DATA_BLOCK "DIH"
{ S7_Optimized_Access := 'FALSE' }
VERSION : 0.1
NON_RETAIN
   STRUCT
      HAD10_AA101_PWR : "DIVAR_HMI";   // Клапан неперевної продувки. (Контроль живлення) {CJF01}
      LAB10_AA001_PWR : "DIVAR_HMI";   // Регулятор рівня в барабані. (Контроль живлення) {CJF01}
      CJF01_SB001_ESTP : "DIVAR_HMI";   // СТОП Шафа SCPU {CJF01}
      CJF01_SB002_ESTP : "DIVAR_HMI";   // СТОП Шафа Пневмоострів {CJF01}
      REZDI_CJF01_MOD11_CH4 : "DIVAR_HMI";   // Резерв DI, рейка CJF01, модуль 11, канал 4 {CJF01}
      HCB10_AA601_SOPN : "DIVAR_HMI";   // Клапан Обдувного апарату №1 (Спрацювання) {CJF01}
      HCB20_AA601_SOPN : "DIVAR_HMI";   // Клапан Обдувного апарату №2 (Спрацювання) {CJF01}
      HCB30_AA601_SOPN : "DIVAR_HMI";   // Клапан Обдувного апарату №3 (Спрацювання) {CJF01}
      HCB40_AA601_SOPN : "DIVAR_HMI";   // Клапан Обдувного апарату №4 (Спрацювання) {CJF01}
      HCB50_AA601_SOPN : "DIVAR_HMI";   // Клапан Обдувного апарату №5 (Спрацювання) {CJF01}
      HCB60_AA601_SOPN : "DIVAR_HMI";   // Клапан Обдувного апарату №6 (Спрацювання) {CJF01}
      HCB70_AA601_SOPN : "DIVAR_HMI";   // Клапан Обдувного апарату №7 (Спрацювання) {CJF01}
      HCB80_AA601_SOPN : "DIVAR_HMI";   // Клапан Обдувного апарату №8 (Спрацювання) {CJF01}
      HCB90_AA601_SOPN : "DIVAR_HMI";   // Клапан Обдувного апарату №9 (Спрацювання) {CJF01}
      HCB100_AA601_SOPN : "DIVAR_HMI";   // Клапан Обдувного апарату №10 (Спрацювання) {CJF01}
      REZDI_CJF01_MOD11_CH15 : "DIVAR_HMI";   // Резерв DI, рейка CJF01, модуль 11, канал 15 {CJF01}
      HLA10_AA151_SOPN : "DIVAR_HMI";   // Шибер первинного повітря №1 (Відкритий) {CJF01}
      HLA10_AA151_SCLS : "DIVAR_HMI";   // Шибер первинного повітря №1 (Закритий) {CJF01}
      HLA10_AA152_SOPN : "DIVAR_HMI";   // Шибер первинного повітря №2 (Відкритий) {CJF01}
      HLA10_AA152_SCLS : "DIVAR_HMI";   // Шибер первинного повітря №2 (Закритий) {CJF01}
      HHB11_SOPN : "DIVAR_HMI";   // Колосники "Поле №1" (Відкритий) {CJF01}
      HHB11_SCLS : "DIVAR_HMI";   // Колосники "Поле №1" (Закритий) {CJF01}
      HHB12_SOPN : "DIVAR_HMI";   // Колосники "Поле №2" (Відкритий) {CJF01}
      HHB12_SCLS : "DIVAR_HMI";   // Колосники "Поле №2" (Закритий) {CJF01}
      HHB13_SOPN : "DIVAR_HMI";   // Колосники "Поле №3" (Відкритий) {CJF01}
      HHB13_SCLS : "DIVAR_HMI";   // Колосники "Поле №3" (Закритий) {CJF01}
      HHB14_SOPN : "DIVAR_HMI";   // Колосники "Поле №4" (Відкритий) {CJF01}
      HHB14_SCLS : "DIVAR_HMI";   // Колосники "Поле №4" (Закритий) {CJF01}
      REZDI_CJF01_MOD12_CH12 : "DIVAR_HMI";   // Резерв DI, рейка CJF01, модуль 12, канал 12 {CJF01}
      REZDI_CJF01_MOD12_CH13 : "DIVAR_HMI";   // Резерв DI, рейка CJF01, модуль 12, канал 13 {CJF01}
      REZDI_CJF01_MOD12_CH14 : "DIVAR_HMI";   // Резерв DI, рейка CJF01, модуль 12, канал 14 {CJF01}
      REZDI_CJF01_MOD12_CH15 : "DIVAR_HMI";   // Резерв DI, рейка CJF01, модуль 12, канал 15 {CJF01}
      HNC10_AF001_PWR : "DIVAR_HMI";   // Димосос ДН1 (Контроль живлення) {CJF06}
      HNC10_AF001_LSTP : "DIVAR_HMI";   // Димосос ДН1 (Кнопка стоп) {CJF06}
      HNC10_AF001_RUN : "DIVAR_HMI";   // Димосос ДН1 (Робота) {CJF06}
      HNC10_AF001_ALM : "DIVAR_HMI";   // Димосос ДН1 (Аварія ПЧ) {CJF06}
      HNC20_AF001_PWR : "DIVAR_HMI";   // Димосос ДН2 (Контроль живлення) {CJF06}
      HNC20_AF001_LSTP : "DIVAR_HMI";   // Димосос ДН2 (Кнопка стоп) {CJF06}
      HNC20_AF001_RUN : "DIVAR_HMI";   // Димосос ДН2 (Робота) {CJF06}
      HNC20_AF001_ALM : "DIVAR_HMI";   // Димосос ДН2 (Аварія ПЧ) {CJF06}
      HLA10_AF001_PWR : "DIVAR_HMI";   // Вентилятор первинного дуття ДВ1 (Контроль живлення) {CJF06}
      HLA10_AF001_LSTP : "DIVAR_HMI";   // Вентилятор первинного дуття ДВ1 (Кнопка стоп) {CJF06}
      HLA10_AF001_RUN : "DIVAR_HMI";   // Вентилятор первинного дуття ДВ1 (Робота) {CJF06}
      HLA10_AF001_ALM : "DIVAR_HMI";   // Вентилятор первинного дуття ДВ1 (Аварія ПЧ) {CJF06}
      HLA20_AF001_PWR : "DIVAR_HMI";   // Вентилятор вторинного дуття ДВ2 (Контроль живлення) {CJF06}
      HLA20_AF001_LSTP : "DIVAR_HMI";   // Вентилятор вторинного дуття ДВ2 (Кнопка стоп) {CJF06}
      HLA20_AF001_RUN : "DIVAR_HMI";   // Вентилятор вторинного дуття ДВ2 (Робота) {CJF06}
      HLA20_AF001_ALM : "DIVAR_HMI";   // Вентилятор вторинного дуття ДВ2 (Аварія ПЧ) {CJF06}
      LAB01_AP001_PWR : "DIVAR_HMI";   // Живильний насос №1 (Контроль живлення) {CJF06}
      LAB01_AP001_LSTP : "DIVAR_HMI";   // Живильний насос №1 (Кнопка стоп) {CJF06}
      LAB01_AP001_RUN : "DIVAR_HMI";   // Живильний насос №1 (Робота) {CJF06}
      LAB01_AP001_ALM : "DIVAR_HMI";   // Живильний насос №1 (Аварія ПЧ) {CJF06}
      LAB02_AP002_PWR : "DIVAR_HMI";   // Живильний насос №2 (Контроль живлення) {CJF06}
      LAB02_AP002_LSTP : "DIVAR_HMI";   // Живильний насос №2 (Кнопка стоп) {CJF06}
      LAB02_AP002_RUN : "DIVAR_HMI";   // Живильний насос №2 (Робота) {CJF06}
      LAB02_AP002_ALM : "DIVAR_HMI";   // Живильний насос №2 (Аварія ПЧ) {CJF06}
      HFB11_AF001_PWR : "DIVAR_HMI";   // Шнек подачі палива №1 (Контроль живлення) {CJF06}
      HFB11_AF001_LSTP : "DIVAR_HMI";   // Шнек подачі палива №1 (Кнопка стоп) {CJF06}
      HFB11_AF001_RUN : "DIVAR_HMI";   // Шнек подачі палива №1 (Робота) {CJF06}
      HFB11_AF001_ALM : "DIVAR_HMI";   // Шнек подачі палива №1 (Аварія ПЧ) {CJF06}
      HFB21_AF001_PWR : "DIVAR_HMI";   // Шнек подачі палива №2 (Контроль живлення) {CJF06}
      HFB21_AF001_LSTP : "DIVAR_HMI";   // Шнек подачі палива №2 (Кнопка стоп) {CJF06}
      HFB21_AF001_RUN : "DIVAR_HMI";   // Шнек подачі палива №2 (Робота) {CJF06}
      HFB21_AF001_ALM : "DIVAR_HMI";   // Шнек подачі палива №2 (Аварія ПЧ) {CJF06}
      HFB12_AF001_PWR : "DIVAR_HMI";   // Транспортер подачі палива №1 (Контроль живлення) {CJF06}
      HFB12_AF001_LSTP : "DIVAR_HMI";   // Транспортер подачі палива №1 (Кнопка стоп) {CJF06}
      HFB12_AF001_RUN : "DIVAR_HMI";   // Транспортер подачі палива №1 (Робота) {CJF06}
      HFB12_AF001_ALM : "DIVAR_HMI";   // Транспортер подачі палива №1 (Аварія ПЧ) {CJF06}
      HFB22_AF001_PWR : "DIVAR_HMI";   // Транспортер подачі палива №2 (Контроль живлення) {CJF06}
      HFB22_AF001_LSTP : "DIVAR_HMI";   // Транспортер подачі палива №2 (Кнопка стоп) {CJF06}
      HFB22_AF001_RUN : "DIVAR_HMI";   // Транспортер подачі палива №2 (Робота) {CJF06}
      HFB22_AF001_ALM : "DIVAR_HMI";   // Транспортер подачі палива №2 (Аварія ПЧ) {CJF06}
      EKG11_AF001_PWR : "DIVAR_HMI";   // Пульсатор (Контроль живлення) {CJF06}
      EKG11_AF001_LSTP : "DIVAR_HMI";   // Пульсатор (Кнопка стоп) {CJF06}
      EKG11_AF001_RUN : "DIVAR_HMI";   // Пульсатор (Робота) {CJF06}
      EKG11_AF001_ALM : "DIVAR_HMI";   // Пульсатор (Аварія ПЧ) {CJF06}
      Rez1_PWR : "DIVAR_HMI";   // Резервний привод ПЧ (Контроль живлення) {CJF06}
      Rez1_LSTP : "DIVAR_HMI";   // Резервний привод ПЧ (Кнопка стоп) {CJF06}
      Rez1_RUN : "DIVAR_HMI";   // Резервний привод ПЧ (Робота) {CJF06}
      Rez1_ALM : "DIVAR_HMI";   // Резервний привод ПЧ (Аварія ПЧ) {CJF06}
      EKG10_AN001_PWR : "DIVAR_HMI";   // Вентилятор закиду палива ВЛ (Контроль живлення) {CJF06}
      EKG10_AN001_LSTP : "DIVAR_HMI";   // Вентилятор закиду палива ВЛ (Кнопка стоп) {CJF06}
      EKG10_AN001_RUN : "DIVAR_HMI";   // Вентилятор закиду палива ВЛ (Робота) {CJF06}
      ETC10_AF001_PWR : "DIVAR_HMI";   // Конвеєр золи скребковий №1 (Контроль живлення) {CJF06}
      ETC10_AF001_LSTP : "DIVAR_HMI";   // Конвеєр золи скребковий №1 (Кнопка стоп) {CJF06}
      ETC10_AF001_RUN : "DIVAR_HMI";   // Конвеєр золи скребковий №1 (Робота) {CJF06}
      ETC01_AF001_PWR : "DIVAR_HMI";   // Конвеєр золи скребковий №2 (Контроль живлення) {CJF06}
      ETC01_AF001_LSTP : "DIVAR_HMI";   // Конвеєр золи скребковий №2 (Кнопка стоп) {CJF06}
      ETC01_AF001_RUN : "DIVAR_HMI";   // Конвеєр золи скребковий №2 (Робота) {CJF06}
      ETC01_AF002_PWR : "DIVAR_HMI";   // Конвеєр золи гвинтовий №3 (Контроль живлення) {CJF06}
      ETC01_AF002_LSTP : "DIVAR_HMI";   // Конвеєр золи гвинтовий №3 (Кнопка стоп) {CJF06}
      ETC01_AF002_RUN : "DIVAR_HMI";   // Конвеєр золи гвинтовий №3 (Робота) {CJF06}
      ETG21_AF001_PWR : "DIVAR_HMI";   // Шлюзовий затвор №1 (Контроль живлення) {CJF06}
      ETG21_AF001_LSTP : "DIVAR_HMI";   // Шлюзовий затвор №1 (Кнопка стоп) {CJF06}
      ETG21_AF001_RUN : "DIVAR_HMI";   // Шлюзовий затвор №1 (Робота) {CJF06}
      ETG22_AF001_PWR : "DIVAR_HMI";   // Шлюзовий затвор №2 (Контроль живлення) {CJF06}
      ETG22_AF001_LSTP : "DIVAR_HMI";   // Шлюзовий затвор №2 (Кнопка стоп) {CJF06}
      ETG22_AF001_RUN : "DIVAR_HMI";   // Шлюзовий затвор №2 (Робота) {CJF06}
      ETG23_AF001_PWR : "DIVAR_HMI";   // Шлюзовий затвор №3 (Контроль живлення) {CJF06}
      ETG23_AF001_LSTP : "DIVAR_HMI";   // Шлюзовий затвор №3 (Кнопка стоп) {CJF06}
      ETG23_AF001_RUN : "DIVAR_HMI";   // Шлюзовий затвор №3 (Робота) {CJF06}
      ETG24_AF001_PWR : "DIVAR_HMI";   // Шлюзовий затвор №4 (Контроль живлення) {CJF06}
      ETG24_AF001_LSTP : "DIVAR_HMI";   // Шлюзовий затвор №4 (Кнопка стоп) {CJF06}
      ETG24_AF001_RUN : "DIVAR_HMI";   // Шлюзовий затвор №4 (Робота) {CJF06}
      ETG31_AF001_PWR : "DIVAR_HMI";   // Шлюзовий затвор №5 (Контроль живлення) {CJF06}
      ETG31_AF001_LSTP : "DIVAR_HMI";   // Шлюзовий затвор №5 (Кнопка стоп) {CJF06}
      ETG31_AF001_RUN : "DIVAR_HMI";   // Шлюзовий затвор №5 (Робота) {CJF06}
      ETG32_AF001_PWR : "DIVAR_HMI";   // Шлюзовий затвор №6 (Контроль живлення) {CJF06}
      ETG32_AF001_LSTP : "DIVAR_HMI";   // Шлюзовий затвор №6 (Кнопка стоп) {CJF06}
      ETG32_AF001_RUN : "DIVAR_HMI";   // Шлюзовий затвор №6 (Робота) {CJF06}
      ETG41_AF001_PWR : "DIVAR_HMI";   // Шлюзовий затвор №7 (Контроль живлення) {CJF06}
      ETG41_AF001_LSTP : "DIVAR_HMI";   // Шлюзовий затвор №7 (Кнопка стоп) {CJF06}
      ETG41_AF001_RUN : "DIVAR_HMI";   // Шлюзовий затвор №7 (Робота) {CJF06}
      ETG51_AF001_PWR : "DIVAR_HMI";   // Шлюзовий затвор №8 (Контроль живлення) {CJF06}
      ETG51_AF001_LSTP : "DIVAR_HMI";   // Шлюзовий затвор №8 (Кнопка стоп) {CJF06}
      ETG51_AF001_RUN : "DIVAR_HMI";   // Шлюзовий затвор №8 (Робота) {CJF06}
      ETG31_AF002_PWR : "DIVAR_HMI";   // Шнек золовидалення №1 (Контроль живлення) {CJF06}
      ETG31_AF002_LSTP : "DIVAR_HMI";   // Шнек золовидалення №1 (Кнопка стоп) {CJF06}
      ETG31_AF002_RUN : "DIVAR_HMI";   // Шнек золовидалення №1 (Робота) {CJF06}
      ETG32_AF002_PWR : "DIVAR_HMI";   // Шнек золовидалення №2 (Контроль живлення) {CJF06}
      ETG32_AF002_LSTP : "DIVAR_HMI";   // Шнек золовидалення №2 (Кнопка стоп) {CJF06}
      ETG32_AF002_RUN : "DIVAR_HMI";   // Шнек золовидалення №2 (Робота) {CJF06}
      ETG51_AF002_PWR : "DIVAR_HMI";   // Шнек золовидалення №3 (Контроль живлення) {CJF06}
      ETG51_AF002_LSTP : "DIVAR_HMI";   // Шнек золовидалення №3 (Кнопка стоп) {CJF06}
      ETG51_AF002_RUN : "DIVAR_HMI";   // Шнек золовидалення №3 (Робота) {CJF06}
      Rez2_PWR : "DIVAR_HMI";   // Резервний привод №2 (Контроль живлення) {CJF06}
      Rez2_LSTP : "DIVAR_HMI";   // Резервний привод №2 (Кнопка стоп) {CJF06}
      Rez2_RUN : "DIVAR_HMI";   // Резервний привод №2 (Робота) {CJF06}
      EBA10_AA101_PWR : "DIVAR_HMI";   // Відсічний затвор №1 (Контроль живлення) {CJF06}
      EBA10_AA101_LSTP : "DIVAR_HMI";   // Відсічний затвор №1 (Кнопка стоп) {CJF06}
      EBA10_AA101_SCLS : "DIVAR_HMI";   // Відсічний затвор №1 (Положення "Закрита") {CJF06}
      EBA10_AA101_SOPN : "DIVAR_HMI";   // Відсічний затвор №1 (Положення "Відкрита") {CJF06}
      EBA20_AA102_PWR : "DIVAR_HMI";   // Відсічний затвор №2 (Контроль живлення) {CJF06}
      EBA20_AA102_LSTP : "DIVAR_HMI";   // Відсічний затвор №2 (Кнопка стоп) {CJF06}
      EBA20_AA102_SCLS : "DIVAR_HMI";   // Відсічний затвор №2 (Положення "Закрита") {CJF06}
      EBA20_AA102_SOPN : "DIVAR_HMI";   // Відсічний затвор №2 (Положення "Відкрита") {CJF06}
      LBA10_AA102_PWR : "DIVAR_HMI";   // ГПЗ (Контроль живлення) {CJF06}
      LBA10_AA102_LSTP : "DIVAR_HMI";   // ГПЗ (Кнопка стоп) {CJF06}
      LBA10_AA102_SCLS : "DIVAR_HMI";   // ГПЗ (Положення "Закрита") {CJF06}
      LBA10_AA102_SOPN : "DIVAR_HMI";   // ГПЗ (Положення "Відкрита") {CJF06}
      REZDI_CJF06_MOD7_CH12 : "DIVAR_HMI";   // Резерв DI, рейка CJF06, модуль 7, канал 12 {CJF06}
      REZDI_CJF06_MOD7_CH13 : "DIVAR_HMI";   // Резерв DI, рейка CJF06, модуль 7, канал 13 {CJF06}
      REZDI_CJF06_MOD7_CH14 : "DIVAR_HMI";   // Резерв DI, рейка CJF06, модуль 7, канал 14 {CJF06}
      REZDI_CJF06_MOD7_CH15 : "DIVAR_HMI";   // Резерв DI, рейка CJF06, модуль 7, канал 15 {CJF06}
      HCB100_AN002_PWR : "DIVAR_HMI";   // Каретка обдувочного апарату №1. (Контроль живлення) {CJF06}
      HCB100_AN002_LSTP : "DIVAR_HMI";   // Каретка обдувочного апарату №1. (Кнопка стоп) {CJF06}
      HCB100_AN002_SOPN : "DIVAR_HMI";   // Каретка обдувочного апарату №1. Положення "введено" {CJF06}
      HCB100_AN002_SCLS : "DIVAR_HMI";   // Каретка обдувочного апарату №1. Положення "виведено" {CJF06}
      HCB00_AN000_PWR : "DIVAR_HMI";   // Обдувні апарати. (Контроль живлення) {CJF06}
      HCB10_AN001_RUN : "DIVAR_HMI";   // Обдувочний апарат №1. (Робота) {CJF06}
      HCB20_AN001_RUN : "DIVAR_HMI";   // Обдувочний апарат №2. (Робота) {CJF06}
      HCB30_AN001_RUN : "DIVAR_HMI";   // Обдувочний апарат №3. (Робота) {CJF06}
      HCB40_AN001_RUN : "DIVAR_HMI";   // Обдувочний апарат №4. (Робота) {CJF06}
      HCB50_AN001_RUN : "DIVAR_HMI";   // Обдувочний апарат №5. (Робота) {CJF06}
      HCB60_AN001_RUN : "DIVAR_HMI";   // Обдувочний апарат №6. (Робота) {CJF06}
      HCB70_AN001_RUN : "DIVAR_HMI";   // Обдувочний апарат №7. (Робота) {CJF06}
      HCB80_AN001_RUN : "DIVAR_HMI";   // Обдувочний апарат №8. (Робота) {CJF06}
      HCB90_AN001_RUN : "DIVAR_HMI";   // Обдувочний апарат №9. (Робота) {CJF06}
      HCB100_AN001_RUN : "DIVAR_HMI";   // Обдувочний апарат №10. (Робота) {CJF06}
      REZDI_CJF06_MOD8_CH15 : "DIVAR_HMI";   // Резерв DI, рейка CJF06, модуль 8, канал 15 {CJF06}
   END_STRUCT;


BEGIN

END_DATA_BLOCK

